PROGRAM MAIN
VAR
END_VAR

END_PROGRAM

(* stored: Version 1.1.0.1
   POU MAIN: Id {e4b2c39d-ef41-4c77-abca-47eb2528416b} *)
